PROGRAM PRG_IM3L0_PPM
VAR
    {attribute 'pytmc' := '
        pv: IM3L0:PPM
        io: io
    '}
    {attribute 'TcLinkTo' := '.fbGige.iIlluminatorINT := TIIB[IM3L0-EL4004]^AO Outputs Channel 1^Analog output;
                              .fbGige.bGigePower := TIIB[IM3L0-EL2004]^Channel 2^Output;
                              .fbPowerMeter.iVoltageINT := TIIB[IM3L0-EL3062]^AI Standard Channel 1^Value;
                              .fbPowerMeter.fbTempSensor.bError := TIIB[IM3L0-EL3314]^TC Inputs Channel 1^Status^Error;
                              .fbPowerMeter.fbTempSensor.bUnderrange := TIIB[IM3L0-EL3314]^TC Inputs Channel 1^Status^Underrange;
                              .fbPowerMeter.fbTempSensor.bOverrange := TIIB[IM3L0-EL3314]^TC Inputs Channel 1^Status^Overrange;
                              .fbPowerMeter.fbTempSensor.iRaw := TIIB[IM3L0-EL3314]^TC Inputs Channel 1^Value;
                              .fbYagTempSensor.bError := TIIB[IM3L0-EL3314]^TC Inputs Channel 2^Status^Error;
                              .fbYagTempSensor.bUnderrange := TIIB[IM3L0-EL3314]^TC Inputs Channel 2^Status^Underrange;
                              .fbYagTempSensor.bOverrange := TIIB[IM3L0-EL3314]^TC Inputs Channel 2^Status^Overrange;
                              .fbYagTempSensor.iRaw := TIIB[IM3L0-EL3314]^TC Inputs Channel 2^Value'}
    fbIM3L0: FB_PPM;

    fbStateSetup: FB_StateSetupHelper;
    stDefault: ST_PositionState := (
        fVelocity := 10,
        bMoveOk := TRUE,
        bValid := TRUE
    );
END_VAR


fbStateSetup(stPositionState:=stDefault, bSetDefault:=TRUE);
fbStateSetup(stPositionState:=fbIM3L0.stOut, fPosition:=-8.40,    sPmpsState:='IM3L0:PPM-OUT');
fbStateSetup(stPositionState:=fbIM3L0.stPower, fPosition:=-47.40, sPmpsState:='IM3L0:PPM-POWERMETER');
fbStateSetup(stPositionState:=fbIM3L0.stYag1, fPosition:=-71.50,  sPmpsState:='IM3L0:PPM-YAG1');
fbStateSetup(stPositionState:=fbIM3L0.stYag2, fPosition:=-97.51,  sPmpsState:='IM3L0:PPM-YAG2');

fbIM3L0(
    fbArbiter := GVL.fbArbiter,
    fbFFHWO := GVL.fbFastFaultOutput1c,
    stYStage := Main.M27,
    sDeviceName := 'IM3L0:PPM',
    sTransitionKey := 'IM3L0:PPM-TRANSITION',
    bEnableMotion := TRUE,
    bEnableBeamParams := TRUE,
    bEnablePositionLimits := TRUE,
    fResponsivity := 0.0506,
);

END_PROGRAM

(* stored: Version 1.1.0.1
   POU PRG_IM3L0_PPM: Id {e4255619-3c3a-488b-9f38-90b77c8df5be}, SpecialFunc None *)
